TYPE ST_InOutputsSTI_EtherCAT_Conveyor :
(**************************************************************************************
 * 	Application		:	BoxControl Framework
 *	Revision		:	$Revision: 354300 $
 *	Revision date	:	$Date: 2015-09-02 12:23:37 +0200 (Mi, 02 Sep 2015) $
 *	Last changed by	:	$Author: d7mangc $
 *	URL				:	$URL: http://almscdc.swisslog.com/repo/SWPD/Development/BoxControlFramework/20_Release/trunk/01_Software/BoxControlFramework/BoxControlFramework/JumpStart/11_Library/10_Application/12_ElementFunctions/01_DUTs/11_Base/ST_TransportData.TcDUT $
 *
 *	Purpose			:	Subsystem transport interface conveyor over EtherCAT
 *
 * ------------------------------------------------------------------------------------
 *	Copyright Swisslog [IP AG], Switzerland. All rights reserved.
 * 
 * ------------------------------------------------------------------------------------
 *	
 * 	Revision History: 
 *
 * 	VERSION			DATE			INITIALS			DESCRIPTION
 *	0.1				01.01.2001		swl					Example
 *
 **************************************************************************************)	
STRUCT
	Watchdog			: BOOL; // Communication supervision 
	eTakeOverState 		: E_TakeOverState; // Takeover state
	eHandOverState 		: E_HandOverState ; // Handover state
	FastSpeedActive		: BOOL; // Fast speed active
	TransportActive		: BOOL; // Transport ongoing
	TU_ID				: STRING(Conveyor.TU_ID_STRINGLENGTH); // TU ID
	Destination			: STRING(Conveyor.POSITION_STRINGLENGTH); // Destination
	AssignmentID		: UDINT; // Assignment ID
END_STRUCT
END_TYPE

(* stored: Version 1.1.0.1, ProductVersion 3.1.4022.12
   DUT ST_InOutputsSTI_EtherCAT_Conveyor: Id {1467d07e-13bf-46bc-b3de-ea894d1e11c8} *)
